// TIA Portal V21 export
DATA_BLOCK "CP01"   // DB23
// stored: InstanceOfName FB614, InstanceOfType FB
"FB614"
   // VAR_INPUT
   //    Simulation : Bool;
   //    Running : Bool;
   //    OnCondition : Bool;
   //    FscInput : Bool;
   //    BypassFscLogic : Bool;
   //    OnDelay : Int;
   //    OffDelay : Int;
   //    CasingDrainDelay : Int;
   // END_VAR
   // VAR_OUTPUT
   //    Output : Bool;
   //    CasingDrainValve : Bool;
   // END_VAR
   // VAR_IN_OUT
   //    Temp1 : DInt;
   //    Temp2 : DInt;
   //    Temp3 : Bool;
   //    Temp4 : Bool;
   //    Temp5 : DInt;
   // END_VAR
   // VAR
   //    OnDelayTimer { S7_SetPoint := 'True'} : TON_TIME;
   //    BypassFSLogicForcefully { S7_SetPoint := 'True'} : TON_TIME;
   //    OffDelayTimer { S7_SetPoint := 'True'} : TON_TIME;
   //    CdTimer { S7_SetPoint := 'True'} : TON_TIME;
   // END_VAR
BEGIN
END_DATA_BLOCK
